(* CODESYS project _02_TaskLocalGVL.task_local_gvl.xml

Project tree, tasks and I/O mapping:
  declarations _02_TaskLocalGVL
*)

// _02_TaskLocalGVL
// [INFO] Task with write access: Task (set manually in CODESYS, not restored by import)
{attribute 'qualified_only'}
VAR_GLOBAL
	iInteger : INT; // [INFO] Integer variable
END_VAR
